TYPE ST_VoltageFeedback :
STRUCT
	voltageFeedback_raw : INT;
END_STRUCT
END_TYPE

(* stored: Version 1.1.0.1, ProductVersion 3.1.4024.11
   DUT ST_VoltageFeedback: Id {b773a86b-33a2-48ab-b571-8d570e3bdc69} *)
